// TIA Portal project "Lab1.4" (V16)

(* hardware
DEVICE "S7-1200 station_1"  S7-1200 Station
   slot 0: "Rack_0"  S7-1200 Rack  Rack  V1.0
   slot 1: "PLC_1"  CPU 1211C AC/DC/Rly  6ES7 211-1BE40-0XB0  V4.4
DEVICE "HMI_1"  KTP700 Basic PN
   slot 0: "HMI_1"  KTP700 Basic PN  6AV2 123-2GB03-0AX0  15.1.0.0
   slot 1: "HMI_RT_1"  KTP700 Basic PN  6AV2 123-2GB03-0AX0  15.1.0.0
   slot 5: "HMI_1.IE_CP_1"  PROFINET Interface  15.0.1.0
      slot 1: "PROFINET Interface_1"  PROFINET Interface
         slot 1: "Port_1"  Port
*)

// ===== PLC "PLC_1"  CPU 1211C AC/DC/Rly =====

VAR_GLOBAL   // PLC tag table "Default tag table"
   "System_Byte" AT %MB1 : Byte;
   "FirstScan" AT %M1.0 : Bool;
   "DiagStatusUpdate" AT %M1.1 : Bool;
   "AlwaysTRUE" AT %M1.2 : Bool;
   "AlwaysFALSE" AT %M1.3 : Bool;
   "Clock_Byte" AT %MB0 : Byte;
   "Clock_10Hz" AT %M0.0 : Bool;
   "Clock_5Hz" AT %M0.1 : Bool;
   "Clock_2.5Hz" AT %M0.2 : Bool;
   "Clock_2Hz" AT %M0.3 : Bool;
   "Clock_1.25Hz" AT %M0.4 : Bool;
   "Clock_1Hz" AT %M0.5 : Bool;
   "Clock_0.625Hz" AT %M0.6 : Bool;
   "Clock_0.5Hz" AT %M0.7 : Bool;
   "PUMP" AT %Q0.0 : Bool;
   "VALVE" AT %Q0.1 : Bool;
END_VAR

DATA_BLOCK "DATA_BLOCK"   // DB1
{ S7_Optimized_Access := 'FALSE' }
VERSION : 0.1
   VAR
      AUTOMATIC_MANUAL : Bool;
      AUTOMATIC_START : Bool;
      AUTOMATIC_STOP : Bool;
      AUTOMATIC_RUN : Bool;
      AUTOMATIC_PUMP : Bool;
      AUTOMATIC_VALVE : Bool;
      HIGH : Bool;
      LOW : Bool := false;
      POSITIVE_SIGNAL_EDGE : Bool;
      TIMER1_DISPLAY : DInt;
      TIMER2_DISPLAY : DInt;
      MANUAL_PUMP_START : Bool;
      MANUAL_PUMP_STOP : Bool;
      MANUAL_PUMP : Bool;
      MANUAL_VALVE_START : Bool;
      MANUAL_VALVE_STOP : Bool;
      MANUAL_VALVE : Bool;
      WATER_LEVEL : DInt;
   END_VAR
BEGIN
END_DATA_BLOCK

// folder: System blocks/Program resources

DATA_BLOCK "TIMER"   // DB2
{ S7_Optimized_Access := 'TRUE' }
AUTHOR : Simatic
FAMILY : IEC
NAME : IEC_TMR
VERSION : 1.0
// stored: InstanceOfName IEC_TIMER
"IEC_TIMER"
BEGIN
END_DATA_BLOCK

DATA_BLOCK "COUNTER_DOWN"   // DB3
{ S7_Optimized_Access := 'TRUE' }
AUTHOR : Simatic
FAMILY : IEC
NAME : CNTR
VERSION : 1.0
// stored: InstanceOfName IEC_COUNTER
"IEC_COUNTER"
BEGIN
END_DATA_BLOCK

DATA_BLOCK "TIMER2"   // DB4
{ S7_Optimized_Access := 'TRUE' }
AUTHOR : Simatic
FAMILY : IEC
NAME : IEC_TMR
VERSION : 1.0
// stored: InstanceOfName IEC_TIMER
"IEC_TIMER"
BEGIN
END_DATA_BLOCK

// folder: (top level)

FUNCTION "AUTOMATIC_MODE" : Void   // FC1, LAD
{ S7_Optimized_Access := 'TRUE' }
VERSION : 0.1
   VAR_TEMP   // added for the SCL form of the ladder/FBD networks
      _w1 : Bool;
   END_VAR
BEGIN

REGION Network 1
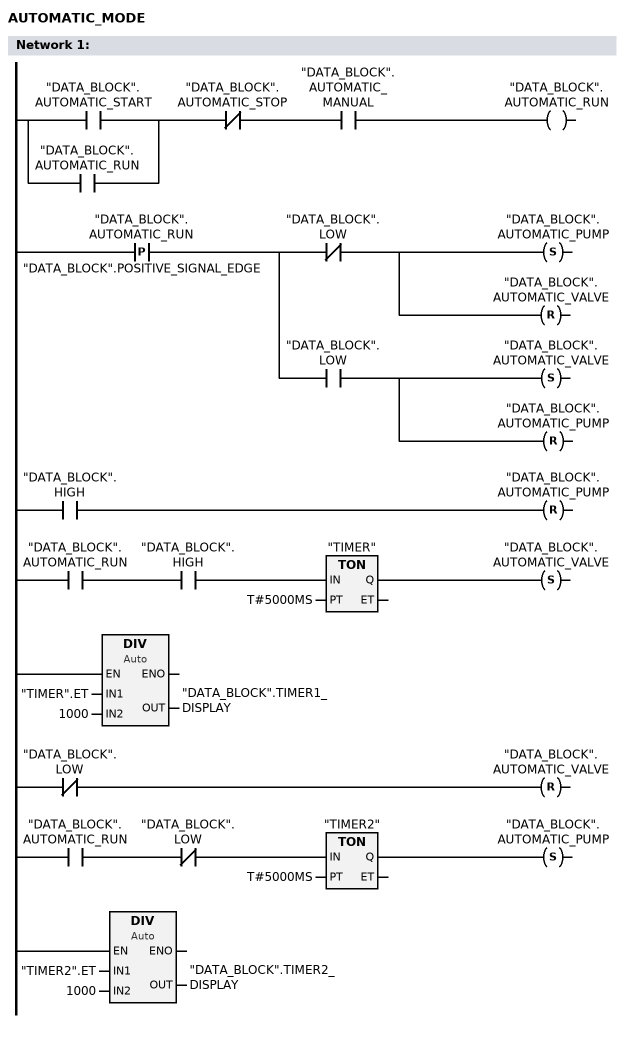
   "DATA_BLOCK".AUTOMATIC_RUN := ("DATA_BLOCK".AUTOMATIC_START OR "DATA_BLOCK".AUTOMATIC_RUN) AND NOT "DATA_BLOCK".AUTOMATIC_STOP AND "DATA_BLOCK".AUTOMATIC_MANUAL;
   #_w1 := "DATA_BLOCK".AUTOMATIC_RUN AND NOT "DATA_BLOCK".POSITIVE_SIGNAL_EDGE;   // rising edge of "DATA_BLOCK".AUTOMATIC_RUN
   "DATA_BLOCK".POSITIVE_SIGNAL_EDGE := "DATA_BLOCK".AUTOMATIC_RUN;
   IF #_w1 AND NOT "DATA_BLOCK".LOW THEN
       "DATA_BLOCK".AUTOMATIC_PUMP := TRUE;
       "DATA_BLOCK".AUTOMATIC_VALVE := FALSE;
   END_IF;
   IF #_w1 AND "DATA_BLOCK".LOW THEN
       "DATA_BLOCK".AUTOMATIC_VALVE := TRUE;
       "DATA_BLOCK".AUTOMATIC_PUMP := FALSE;
   END_IF;
   IF "DATA_BLOCK".HIGH THEN "DATA_BLOCK".AUTOMATIC_PUMP := FALSE; END_IF;
   "TIMER".TON(IN := "DATA_BLOCK".AUTOMATIC_RUN AND "DATA_BLOCK".HIGH, PT := T#5000MS);
   IF "TIMER".Q THEN "DATA_BLOCK".AUTOMATIC_VALVE := TRUE; END_IF;
   "DATA_BLOCK".TIMER1_DISPLAY := "TIMER".ET / 1000;
   IF NOT "DATA_BLOCK".LOW THEN "DATA_BLOCK".AUTOMATIC_VALVE := FALSE; END_IF;
   "TIMER2".TON(IN := "DATA_BLOCK".AUTOMATIC_RUN AND NOT "DATA_BLOCK".LOW, PT := T#5000MS);
   IF "TIMER2".Q THEN "DATA_BLOCK".AUTOMATIC_PUMP := TRUE; END_IF;
   "DATA_BLOCK".TIMER2_DISPLAY := "TIMER2".ET / 1000;
END_REGION
END_FUNCTION

FUNCTION "MANUAL_MODE" : Void   // FC2, LAD
{ S7_Optimized_Access := 'TRUE' }
VERSION : 0.1
BEGIN

REGION Network 1
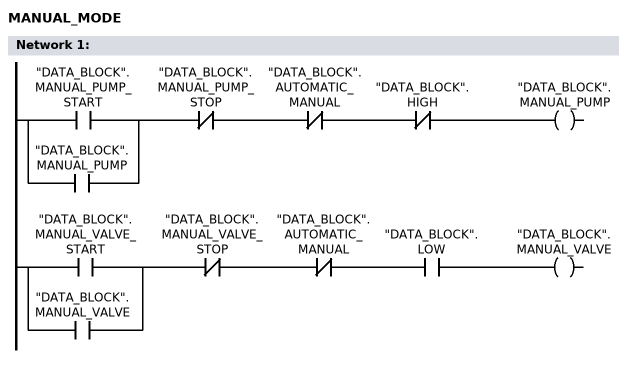
   RUNG wire#powerrail
      Contact( "DATA_BLOCK".MANUAL_PUMP_START )
      wire#w1
      I_Contact( "DATA_BLOCK".MANUAL_PUMP_STOP )
      I_Contact( "DATA_BLOCK".AUTOMATIC_MANUAL )
      I_Contact( "DATA_BLOCK".HIGH )
      Coil( "DATA_BLOCK".MANUAL_PUMP )
   END_RUNG
   RUNG wire#powerrail
      Contact( "DATA_BLOCK".MANUAL_PUMP )
   END_RUNG wire#w1
   RUNG wire#powerrail
      Contact( "DATA_BLOCK".MANUAL_VALVE_START )
      wire#w2
      I_Contact( "DATA_BLOCK".MANUAL_VALVE_STOP )
      I_Contact( "DATA_BLOCK".AUTOMATIC_MANUAL )
      Contact( "DATA_BLOCK".LOW )
      Coil( "DATA_BLOCK".MANUAL_VALVE )
   END_RUNG
   RUNG wire#powerrail
      Contact( "DATA_BLOCK".MANUAL_VALVE )
   END_RUNG wire#w2
   // the same network as SCL:
   "DATA_BLOCK".MANUAL_PUMP := ("DATA_BLOCK".MANUAL_PUMP_START OR "DATA_BLOCK".MANUAL_PUMP) AND NOT "DATA_BLOCK".MANUAL_PUMP_STOP AND NOT "DATA_BLOCK".AUTOMATIC_MANUAL AND NOT "DATA_BLOCK".HIGH;
   "DATA_BLOCK".MANUAL_VALVE := ("DATA_BLOCK".MANUAL_VALVE_START OR "DATA_BLOCK".MANUAL_VALVE) AND NOT "DATA_BLOCK".MANUAL_VALVE_STOP AND NOT "DATA_BLOCK".AUTOMATIC_MANUAL AND "DATA_BLOCK".LOW;
END_REGION
END_FUNCTION

FUNCTION "MAP OUTPUT" : Void   // FC3, LAD
{ S7_Optimized_Access := 'TRUE' }
VERSION : 0.1
BEGIN

REGION Network 1
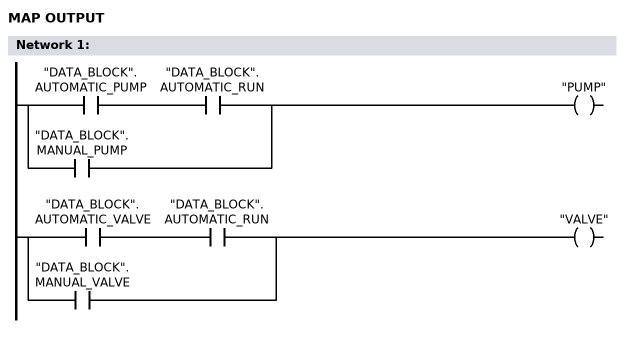
   RUNG wire#powerrail
      Contact( "DATA_BLOCK".AUTOMATIC_PUMP )
      Contact( "DATA_BLOCK".AUTOMATIC_RUN )
      wire#w1
      Coil( "PUMP" )
   END_RUNG
   RUNG wire#powerrail
      Contact( "DATA_BLOCK".MANUAL_PUMP )
   END_RUNG wire#w1
   RUNG wire#powerrail
      Contact( "DATA_BLOCK".AUTOMATIC_VALVE )
      Contact( "DATA_BLOCK".AUTOMATIC_RUN )
      wire#w2
      Coil( "VALVE" )
   END_RUNG
   RUNG wire#powerrail
      Contact( "DATA_BLOCK".MANUAL_VALVE )
   END_RUNG wire#w2
   // the same network as SCL:
   "PUMP" := ("DATA_BLOCK".AUTOMATIC_PUMP AND "DATA_BLOCK".AUTOMATIC_RUN) OR "DATA_BLOCK".MANUAL_PUMP;
   "VALVE" := ("DATA_BLOCK".AUTOMATIC_VALVE AND "DATA_BLOCK".AUTOMATIC_RUN) OR "DATA_BLOCK".MANUAL_VALVE;
END_REGION
END_FUNCTION

FUNCTION "HMI Display" : Void   // FC4, LAD
{ S7_Optimized_Access := 'TRUE' }
VERSION : 0.1
BEGIN

REGION Network 1
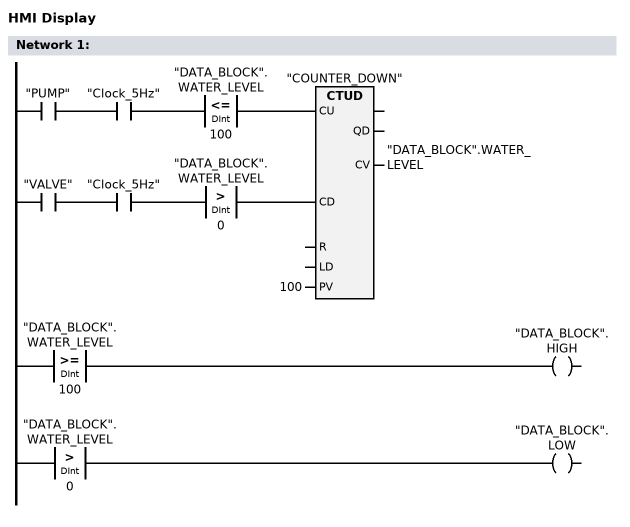
   "COUNTER_DOWN".CTUD(CU := "PUMP" AND "Clock_5Hz" AND ("DATA_BLOCK".WATER_LEVEL <= 100),
                       CD := "VALVE" AND "Clock_5Hz" AND ("DATA_BLOCK".WATER_LEVEL > 0),
                       PV := 100,
                       CV => "DATA_BLOCK".WATER_LEVEL);
   "DATA_BLOCK".HIGH := "DATA_BLOCK".WATER_LEVEL >= 100;
   "DATA_BLOCK".LOW := "DATA_BLOCK".WATER_LEVEL > 0;
END_REGION
END_FUNCTION

ORGANIZATION_BLOCK "Main"   // OB1, LAD, ProgramCycle
TITLE = "Main Program Sweep (Cycle)"
{ S7_Optimized_Access := 'TRUE' }
VERSION : 0.1
   VAR_INPUT
      Initial_Call : Bool;   // Initial call of this OB
      Remanence : Bool;   // =True, if remanent data are available
   END_VAR
BEGIN

REGION Network 1
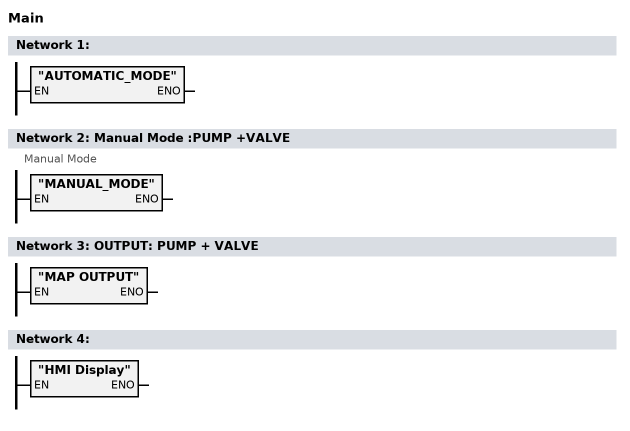
   RUNG wire#powerrail
      "AUTOMATIC_MODE"()
   END_RUNG
   // the same network as SCL:
   "AUTOMATIC_MODE"();
END_REGION

REGION Network 2: Manual Mode :PUMP +VALVE
   // Manual Mode
   RUNG wire#powerrail
      "MANUAL_MODE"()
   END_RUNG
   // the same network as SCL:
   "MANUAL_MODE"();
END_REGION

REGION Network 3: OUTPUT: PUMP + VALVE
   RUNG wire#powerrail
      "MAP OUTPUT"()
   END_RUNG
   // the same network as SCL:
   "MAP OUTPUT"();
END_REGION

REGION Network 4
   RUNG wire#powerrail
      "HMI Display"()
   END_RUNG
   // the same network as SCL:
   "HMI Display"();
END_REGION
END_ORGANIZATION_BLOCK

(* ===== HMI "HMI_RT_1" =====
system functions are stored by id; their names below are inferred from use
connection "HMI_Connection_1": ETHERNET, SMART_S7_1200_OMS
connection "HMI_Connection_2": ETHERNET, SMART_S7_1200_OMS

HMI tags "Default tag table"
   "DATA_BLOCK_AUTOMATIC_MANUAL" : Bool = PLC "DATA_BLOCK".AUTOMATIC_MANUAL AT %DB1.DBX0.0, 1 s
   "DATA_BLOCK_AUTOMATIC_START" : Bool = PLC "DATA_BLOCK".AUTOMATIC_START AT %DB1.DBX0.1, 1 s
   "DATA_BLOCK_AUTOMATIC_STOP" : Bool = PLC "DATA_BLOCK".AUTOMATIC_STOP AT %DB1.DBX0.2, 1 s
   "DATA_BLOCK_AUTOMATIC_RUN" : Bool = PLC "DATA_BLOCK".AUTOMATIC_RUN AT %DB1.DBX0.3, 1 s
   "DATA_BLOCK_AUTOMATIC_PUMP" : Bool = PLC "DATA_BLOCK".AUTOMATIC_PUMP AT %DB1.DBX0.4, 1 s
   "DATA_BLOCK_AUTOMATIC_VALVE" : Bool = PLC "DATA_BLOCK".AUTOMATIC_VALVE AT %DB1.DBX0.5, 1 s
   "DATA_BLOCK_HIGH" : Bool = PLC "DATA_BLOCK".HIGH AT %DB1.DBX0.6, 1 s
   "DATA_BLOCK_LOW" : Bool = PLC "DATA_BLOCK".LOW AT %DB1.DBX0.7, 1 s
   "DATA_BLOCK_POSITIVE_SIGNAL_EDGE" : Bool = PLC "DATA_BLOCK".POSITIVE_SIGNAL_EDGE AT %DB1.DBX1.0, 1 s
   "DATA_BLOCK_TIMER1_DISPLAY" : DInt = PLC "DATA_BLOCK".TIMER1_DISPLAY AT %DB1.DBD2, 1 s
   "DATA_BLOCK_TIMER2_DISPLAY" : DInt = PLC "DATA_BLOCK".TIMER2_DISPLAY AT %DB1.DBD6, 1 s
   "DATA_BLOCK_MANUAL_PUMP_START" : Bool = PLC "DATA_BLOCK".MANUAL_PUMP_START AT %DB1.DBX10.0, 1 s
   "DATA_BLOCK_MANUAL_PUMP_STOP" : Bool = PLC "DATA_BLOCK".MANUAL_PUMP_STOP AT %DB1.DBX10.1, 1 s
   "DATA_BLOCK_MANUAL_PUMP" : Bool = PLC "DATA_BLOCK".MANUAL_PUMP AT %DB1.DBX10.2, 1 s
   "DATA_BLOCK_MANUAL_VALVE_START" : Bool = PLC "DATA_BLOCK".MANUAL_VALVE_START AT %DB1.DBX10.3, 1 s
   "DATA_BLOCK_MANUAL_VALVE_STOP" : Bool = PLC "DATA_BLOCK".MANUAL_VALVE_STOP AT %DB1.DBX10.4, 1 s
   "DATA_BLOCK_MANUAL_VALVE" : Bool = PLC "DATA_BLOCK".MANUAL_VALVE AT %DB1.DBX10.5, 1 s
   "DATA_BLOCK_WATER_LEVEL" : DInt = PLC "DATA_BLOCK".WATER_LEVEL AT %DB1.DBD12, 1 s
   "VALVE" : Bool = PLC VALVE AT %Q0.1, 1 s
   "PUMP" : Bool = PLC PUMP AT %Q0.0, 1 s

screen "Root screen" 800x480, template "Template_1"
   GraphicView "Graphic view_5" at 429,0 size 176x70; Picture "Graphic_10"
   GraphicView "Graphic view_2" at 602,0 size 73x71; Picture "Graphic_12"
   GraphicView "Graphic view_1" at 597,329 size 103x56; Picture "Graphic_6"
   GraphicView "Graphic view_3" at 585,59 size 111x305; Picture "Graphic_8"
   Button "HmiScreenItemData_1" at 36,36 size 159x47; TextOff 'System screens'; PictureOff "Navigates to System screens for KTP700 Basic+ PN 16.0.0.0"; PictureOn "Navigates to System screens for KTP700 Basic+ PN 16.0.0.0"
      on Release: ActivateScreen("System screens", 0)
   Switch "Switch_1" at 47,191 size 159x52; CaptionText 'Switch'; TextOff 'AUTO'; TextOn 'MANUAL'
      on SwitchOn: InvertBit("DATA_BLOCK_AUTOMATIC_MANUAL")
      on SwitchOff: InvertBit("DATA_BLOCK_AUTOMATIC_MANUAL")
   Circle "Circle_1" at 55,123 size 60x60
      Appearance <- "DATA_BLOCK_AUTOMATIC_MANUAL"
   Circle "Circle_2" at 124,123 size 60x60
      Appearance <- "DATA_BLOCK_AUTOMATIC_MANUAL"
   TextField "Text field_1" at 130,94 size 44x23; Text 'Auto'
   TextField "Text field_2" at 55,98 size 69x23; Text 'Manual'
   TextField "Text field_3" at 46,296 size 123x27; Text 'AUTOMATIC'
   Circle "Circle_3" at 184,287 size 48x48
      Appearance <- "DATA_BLOCK_AUTOMATIC_RUN"
   Button "Button_1" at 46,340 size 96x32; TextOff 'START'
      on Press: SetBit("DATA_BLOCK_AUTOMATIC_START")
      on Release: ResetBit("DATA_BLOCK_AUTOMATIC_START")
      Appearance <- "DATA_BLOCK_AUTOMATIC_START"
   Button "Button_2" at 47,389 size 96x32; TextOff 'STOP'
      on Press: SetBit("DATA_BLOCK_AUTOMATIC_STOP")
      on Release: ResetBit("DATA_BLOCK_AUTOMATIC_STOP")
      Appearance <- "DATA_BLOCK_AUTOMATIC_STOP"
   TextField "Text field_4" at 299,123 size 60x27; Text 'PUMP'
      Appearance <- "PUMP"
   Circle "Circle_4" at 361,115 size 48x48
      Appearance <- "PUMP"
   TextField "Text field_5" at 575,396 size 67x27; Text 'VALVE'
      Appearance <- "VALVE"
   Circle "Circle_5" at 648,383 size 48x48
      Appearance <- "VALVE"
   IOField "I/O field_1" at 301,234 size 96x32; FormatPattern s9999999999
      ProcessValue <- "DATA_BLOCK_TIMER1_DISPLAY"
   IOField "I/O field_2" at 436,364 size 96x32; FormatPattern s9999999999
      ProcessValue <- "DATA_BLOCK_TIMER2_DISPLAY"
   TextField "Text field_6" at 301,207 size 87x27; Text 'TIMER 1'
      Appearance <- "VALVE"
   TextField "Text field_7" at 436,337 size 87x27; Text 'TIMER 2'
      Appearance <- "VALVE"
   Bar "Bar_1" at 590,132 size 98x134; MinimumValue 0; MaximumValue 100
      ProcessValue <- "DATA_BLOCK_WATER_LEVEL"
   GraphicView "Graphic view_4" at 293,14 size 143x109; Picture "Graphic_5"
   Button "Button_3" at 249,166 size 96x32; TextOff 'START'
      on Press: SetBit("DATA_BLOCK_MANUAL_PUMP_START")
      on Release: ResetBit("DATA_BLOCK_MANUAL_PUMP_START")
      Appearance <- "DATA_BLOCK_MANUAL_PUMP_START"
   Button "Button_4" at 359,167 size 96x32; TextOff 'STOP'
      on Press: SetBit("DATA_BLOCK_MANUAL_PUMP_STOP")
      on Release: ResetBit("DATA_BLOCK_MANUAL_PUMP_STOP")
      Appearance <- "DATA_BLOCK_MANUAL_PUMP_STOP"
   Button "Button_5" at 538,430 size 96x32; TextOff 'START'
      on Press: SetBit("DATA_BLOCK_MANUAL_VALVE_START")
      on Release: ResetBit("DATA_BLOCK_MANUAL_VALVE_START")
      Appearance <- "DATA_BLOCK_MANUAL_VALVE_START"
   Button "Button_6" at 648,431 size 96x32; TextOff 'STOP'
      on Press: SetBit("DATA_BLOCK_MANUAL_VALVE_STOP")
      on Release: ResetBit("DATA_BLOCK_MANUAL_VALVE_STOP")
      Appearance <- "DATA_BLOCK_MANUAL_VALVE_STOP"

screen "System screens" 800x480, template "Template_1"
   Button "Back" at 1,1 size 159x47; TextOff 'Back'
      on Release: ActivateScreen("Root screen", 0)
   Button "HmiScreenItemData" at 36,95 size 159x47; TextOff 'SIMATIC PLC system diagnos...'; PictureOff "Navigates to SIMATIC PLC system diagnostics for KTP700 Basic+ PN 16.0.0.0"; PictureOn "Navigates to SIMATIC PLC system diagnostics for KTP700 Basic+ PN 16.0.0.0"
      on Release: ActivateScreen("SIMATIC PLC system diagnostics", 0)
   Button "HmiScreenItemData_1" at 36,154 size 159x47; TextOff 'Project information'; PictureOff "Navigates to Project information for KTP700 Basic+ PN 16.0.0.0"; PictureOn "Navigates to Project information for KTP700 Basic+ PN 16.0.0.0"
      on Release: ActivateScreen("Project information", 0)
   Button "HmiScreenItemData_2" at 36,213 size 159x47; TextOff 'User administration'; PictureOff "Navigates to User administration for KTP700 Basic+ PN 16.0.0.0"; PictureOn "Navigates to User administration for KTP700 Basic+ PN 16.0.0.0"
      on Release: ActivateScreen("User administration", 0)
   Button "HmiScreenItemData_3" at 36,272 size 159x47; TextOff 'System information'; PictureOff "Navigates to System information for KTP700 Basic+ PN 16.0.0.0"; PictureOn "Navigates to System information for KTP700 Basic+ PN 16.0.0.0"
      on Release: ActivateScreen("System information", 0)
   Button "HmiScreenItemData_4" at 36,331 size 159x47; TextOff 'Different jobs'; PictureOff "Navigates to Different jobs for KTP700 Basic+ PN 16.0.0.0"; PictureOn "Navigates to Different jobs for KTP700 Basic+ PN 16.0.0.0"
      on Release: ActivateScreen("Different jobs", 0)

screen "SIMATIC PLC system diagnostics" 800x480, template "Template_1"
   SysDiagControl "HmiScreenItemData" at 1,49 size 796x423
   Button "Back" at 1,1 size 159x47; TextOff 'Back'
      on Release: ActivateScreen("System screens", 0)

screen "Project information" 800x480, template "Template_1"
   TextField "HmiScreenItemData" at 35,51 size 171x28; Text 'Project name:'
   TextField "HmiScreenItemData_1" at 241,51 size 524x28; Text 'Lab1.4'
   TextField "HmiScreenItemData_2" at 35,81 size 171x28; Text 'Created on:'
   TextField "HmiScreenItemData_3" at 241,81 size 524x28; Text '6/9/2026 9:58:01 AM'
   TextField "HmiScreenItemData_4" at 35,111 size 171x28; Text 'Author:'
   TextField "HmiScreenItemData_5" at 241,111 size 524x28; Text 'Khoa'
   TextField "HmiScreenItemData_6" at 35,141 size 171x28; Text 'Description:'
   TextField "HmiScreenItemData_7" at 241,141 size 524x28; Text '(not configured)'
   Button "Back" at 1,1 size 159x47; TextOff 'Back'
      on Release: ActivateScreen("System screens", 0)

screen "User administration" 800x480, template "Template_1"
   UserView "HmiScreenItemData" at 1,49 size 796x423
   Button "Back" at 1,1 size 159x47; TextOff 'Back'
      on Release: ActivateScreen("System screens", 0)

screen "System information" 800x480, template "Template_1"
   TextField "HmiScreenItemData" at 35,51 size 171x28; Text 'HMI device type:'
   TextField "HmiScreenItemData_1" at 241,51 size 524x28; Text 'KTP700 Basic+ PN 16.0.0.0'
   TextField "HmiScreenItemData_2" at 35,81 size 171x28; Text 'Connection:'
   TextField "HmiScreenItemData_3" at 241,81 size 524x28; Text 'PROFINET (X1)'
   TextField "HmiScreenItemData_4" at 35,111 size 171x28; Text 'PLC:'
   TextField "HmiScreenItemData_5" at 241,111 size 524x28; Text 'SIMATIC S7 1200'
   Button "Back" at 1,1 size 159x47; TextOff 'Back'
      on Release: ActivateScreen("System screens", 0)

screen "Different jobs" 800x480, template "Template_1"
   Button "Online" at 36,95 size 159x47; TextOff 'Online'
      on Release: function_bb44b551(0)
   Button "Offline" at 36,154 size 159x47; TextOff 'Offline'
      on Release: function_bb44b551(1)
   Button "Transfer" at 36,213 size 159x47; TextOff 'Transfer'
      on Release: function_bb44b551(2)
   Button "Toggle language" at 36,272 size 159x47; TextOff 'Toggle language'
      on Release: function_fb9197e8(-1)
   Button "Stop Runtime" at 36,331 size 159x47; TextOff 'Stop Runtime'
      on Release: StopRuntime(0)
   Button "Back" at 1,1 size 159x47; TextOff 'Back'
      on Release: ActivateScreen("System screens", 0)
*)